// TwinCAT 3 PLC project Reporting_PLC
// ProgramVersion: 3.1.4026.13
// libraries:
//   Tc2_ControllerToolbox, * (Beckhoff Automation GmbH)
//   Tc2_Standard, * (Beckhoff Automation GmbH)
//   Tc2_System, * (Beckhoff Automation GmbH)
// project tree:
//   / PlcTask.TcTTO
//   POUs/ FB_TableData.TcPOU, MAIN.TcPOU
// real-time tasks:
//   TASK PlcTask: cycle T#10ms, priority 20, ADS port 350

CONFIGURATION Reporting_PLC
    RESOURCE PLC ON TwinCAT3
        TASK PlcTask(INTERVAL := T#10ms, PRIORITY := 20);
        PROGRAM MAIN WITH PlcTask : MAIN;
    END_RESOURCE
END_CONFIGURATION

// ---- POUs/MAIN.TcPOU
PROGRAM MAIN
VAR
	{ attribute 'TcHmiSymbol.AddSymbol' }
	_sProjectName	: STRING := 'Reporting sample project';
	{ attribute 'TcHmiSymbol.AddSymbol' }
	_aTableData		: ARRAY[0..10] OF FB_TableData;
	{ attribute 'TcHmiSymbol.AddSymbol' }
	_temperature	: LREAL;
	
	_fbSinus		: FB_CTRL_SIGNAL_GENERATOR := (
						eState 			:= E_CTRL_STATE.eCTRL_STATE_ACTIVE);
	_stSinusParams	: ST_CTRL_SIGNAL_GENERATOR_PARAMS := (
						tCtrlCycleTime 	:= TIME#200MS, 
						tTaskCycleTime 	:= TIME#200MS, 
						eSignalType 	:= E_CTRL_SIGNAL_TYPE.eCTRL_SINUS, 
						tCylceDuration 	:= TIME#40S, 
						fAmplitude 		:= 30, 
						fOffset 		:= 5, 
						tStart 			:= TIME#20MS);
						
	_i				: USINT;
END_VAR


FOR _i := 0 TO 10 DO
	_aTableData[_i].nId := _i;
	_aTableData[_i].sName := CONCAT ('Hello World ',TO_STRING(_i));
	_aTableData[_i].nValue := _i * 1.35;
END_FOR

_fbSinus(
	stParams	:= _stSinusParams);
	
_temperature	:= _fbSinus.fOut;

END_PROGRAM

// ---- POUs/FB_TableData.TcPOU
FUNCTION_BLOCK FB_TableData
VAR_INPUT
	nId		: USINT;
	sName	: STRING;
	nValue	: LREAL;
END_VAR
VAR_OUTPUT
END_VAR
VAR
END_VAR

END_FUNCTION_BLOCK
